FUNCTION_BLOCK CylControlAdpOL (* Composite Function Block Type *)
  (* Standard: 61499-2 *)
  (* Version 0.0, 7/14/2023, valeriy, nxtControl GmBH, template *)
  PACKAGE Main;
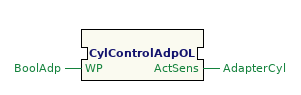
  SOCKETS
    WP : BoolAdp;
  END_SOCKETS
  PLUGS
    ActSens : AdapterCyl;
  END_PLUGS
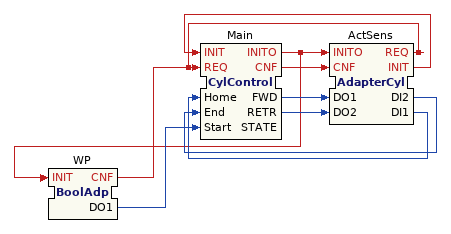
  FBS
    Main : CylControl;
  END_FBS
  EVENT_CONNECTIONS
    WP.CNF TO Main.REQ;
    Main.INITO TO ActSens.INITO;
    Main.CNF TO ActSens.CNF;
    Main.INITO TO WP.INIT;
    ActSens.REQ TO Main.REQ;
    ActSens.INIT TO Main.INIT;
  END_CONNECTIONS
  DATA_CONNECTIONS
    WP.DO1 TO Main.Start;
    Main.FWD TO ActSens.DO1;
    Main.RETR TO ActSens.DO2;
    ActSens.DI2 TO Main.End;
    ActSens.DI1 TO Main.Home;
  END_CONNECTIONS
END_FUNCTION_BLOCK
